{attribute addProperty BoxType "EL9221-4030-0018"}
{attribute addProperty Id "ControlAT %Q*Control_6B063D74162"}
{attribute addProperty CRC "4080052502"}
{attribute addProperty SizeInBites "16"}
{attribute addProperty SizeInBytes "2"}
TYPE OCP_Outputs_F330A916 :
STRUCT
	{attribute addProperty Name "Control"}
	Control AT %Q* : Control_6B063D74;
END_STRUCT
END_TYPE

(* stored: Version 1.2.0.0, ProductVersion 3.1.4024.9
   DUT OCP_Outputs_F330A916: Id {732600ac-1dee-4c79-bfa3-81a7d364e819} *)
